FUNCTION_BLOCK XSPACE (* A spacer object with center and edge labels *)
  (* Standard: 61499-1 *)
  (* Version 0.1, 2004-09-09, JHC, Rockwell Automation, Set DIA initial value to zero. *)
  (* Version 0.0, 2000-04-26, JHC, Rockwell Automation *)
  (* Compiler header: package fb.rt.hmi; *)
  (* Compiler Java IBM VisualAge 3.0 *)
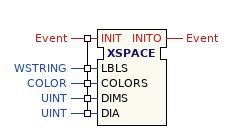
  EVENT_INPUT
    INIT WITH LBLS, COLORS, DIMS, DIA; (* Initialize *)
  END_EVENT
  EVENT_OUTPUT
    INITO; (* Initialization Confirm *)
  END_EVENT
  VAR_INPUT
    LBLS : WSTRING; (* Labels:{Left,Top,Right,Bottom,Center} *)
    COLORS : COLOR; (* {Foreground,Background} *)
    DIMS : UINT; (* {Width,Height}in Diameters *)
    DIA : UINT; (* Diameter dimension *)
  END_VAR
END_FUNCTION_BLOCK
